TYPE ST_StepperMotorCommand :
STRUCT
	Homing : BOOL;
	Command : LREAL;
	Position : LREAL;
	Homed : BOOL;
END_STRUCT
END_TYPE

(* stored: Version 1.1.0.1, ProductVersion 3.1.4026.11
   DUT ST_StepperMotorCommand: Id {6e8dec26-6f30-4f23-8fa3-4e0f61826fd7} *)
